// TIA Portal V19 export
DATA_BLOCK "TestInterConnLPythagorean"   // DB10001
{ S7_Optimized_Access := 'TRUE' }
// #@AutoGenerated
// stored: MemoryReserve 100
   VAR
      "a" : Real;
      "b" : Real;
      c : Real;
      valid : Bool;
   END_VAR
BEGIN
END_DATA_BLOCK
